// TwinCAT 3 PLC project TestPLC
// ProgramVersion: 3.1.4023.0
// libraries:
//   Tc2_Standard, * (Beckhoff Automation GmbH)
//   Tc2_System, * (Beckhoff Automation GmbH)
//   Tc3_Module, * (Beckhoff Automation GmbH)
// project tree:
//   DUTs/ TestStruct.TcDUT
//   GVLs/ GVL.TcGVL
//   / PlcTask.TcTTO
//   POUs/ MAIN.TcPOU
// real-time tasks:
//   TASK PlcTask: cycle T#10ms, priority 20, ADS port 350

CONFIGURATION TestPLC
    RESOURCE PLC ON TwinCAT3
        TASK PlcTask(INTERVAL := T#10ms, PRIORITY := 20);
        PROGRAM MAIN WITH PlcTask : MAIN;
    END_RESOURCE
END_CONFIGURATION

// ---- DUTs/TestStruct.TcDUT
TYPE TestStruct :
STRUCT
	iVal : DINT := 0;
	fVal : REAL := 0.0;
	sVal : STRING := '';
END_STRUCT
END_TYPE

// ---- GVLs/GVL.TcGVL
{attribute 'qualified_only'}
VAR_GLOBAL
	
	// PLC structure for testing type resolution in ADS client
	PlcStruct : TestStruct;
	
	// Vars for client global event handler
	iEventData1 : DINT := 1;
	fEventData2 : REAL := 3.14;
	
	// Var for client custom event handler
	iCustomEvent : DINT := 2;
	
END_VAR

// ---- POUs/MAIN.TcPOU
PROGRAM MAIN
VAR
END_VAR

END_PROGRAM
